// Block: IPC_Com_Channel_LOG_PARAMETRI

DATA_BLOCK IPC_Com_Channel_LOG_PARAMETRI
VERSION : 0.1
   NON_RETAIN
   VAR
      RECEIVE : Struct
         ack : DInt;
         msg : IPC_Msg_Log_PAR;
      END_STRUCT;
      SEND : Struct
         ack : DInt;
         msg : IPC_Msg_Log_PAR;
      END_STRUCT;
   END_VAR

BEGIN
   // No initialization required
END_DATA_BLOCK
